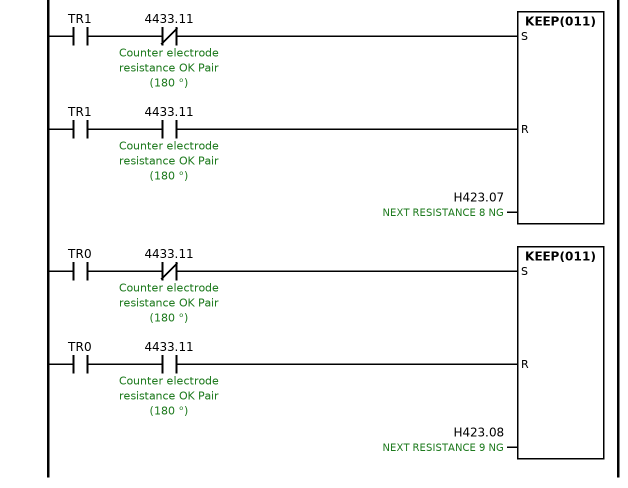
; [picture p408: MainProgram / ST07_RESISTANSE_UNIT, rungs 120-120]
; rung 120
LD 4433.08  ; Counter electrode resistance measurement (180 °)
OUT TR0
AND 4421.01  ; Number of counter electrode resistance 1 *
OUT TR1
ANDNOT 4433.11  ; Counter electrode resistance OK Pair (180 °)
LD TR1
AND 4433.11  ; Counter electrode resistance OK Pair (180 °)
KEEP(011) H423.00  ; NEXT RESISTANCE 1 NG
LD TR0
AND 4421.02  ; Number of adjacent resistances * 2
OUT TR1
ANDNOT 4433.11  ; Counter electrode resistance OK Pair (180 °)
LD TR1
AND 4433.11  ; Counter electrode resistance OK Pair (180 °)
KEEP(011) H423.01  ; NEXT RESISTANCE 2 NG
LD TR0
AND 4421.03  ; Number of adjacent resistances * 3
OUT TR1
ANDNOT 4433.11  ; Counter electrode resistance OK Pair (180 °)
LD TR1
AND 4433.11  ; Counter electrode resistance OK Pair (180 °)
KEEP(011) H423.02  ; NEXT RESISTANCE 3 NG
LD TR0
AND 4421.04  ; Number of adjacent resistances * 4
OUT TR1
ANDNOT 4433.11  ; Counter electrode resistance OK Pair (180 °)
LD TR1
AND 4433.11  ; Counter electrode resistance OK Pair (180 °)
KEEP(011) H423.03  ; NEXT RESISTANCE 4 NG
LD TR0
AND 4421.05  ; Number of adjacent resistances * 5
OUT TR1
ANDNOT 4433.11  ; Counter electrode resistance OK Pair (180 °)
LD TR1
AND 4433.11  ; Counter electrode resistance OK Pair (180 °)
KEEP(011) H423.04  ; NEXT RESISTANCE 5 NG
LD TR0
AND 4421.06  ; Number of adjacent resistances * 6
OUT TR1
ANDNOT 4433.11  ; Counter electrode resistance OK Pair (180 °)
LD TR1
AND 4433.11  ; Counter electrode resistance OK Pair (180 °)
KEEP(011) H423.05  ; NEXT RESISTANCE 6 NG
LD TR0
AND 4421.07  ; Number of adjacent resistances * 7
OUT TR1
ANDNOT 4433.11  ; Counter electrode resistance OK Pair (180 °)
LD TR1
AND 4433.11  ; Counter electrode resistance OK Pair (180 °)
KEEP(011) H423.06  ; NEXT RESISTANCE 7 NG
LD TR0
AND 4421.08  ; Number of adjacent resistances * 8
OUT TR1
ANDNOT 4433.11  ; Counter electrode resistance OK Pair (180 °)
LD TR1
AND 4433.11  ; Counter electrode resistance OK Pair (180 °)
KEEP(011) H423.07  ; NEXT RESISTANCE 8 NG
LD TR0
AND 4421.09  ; Number of adjacent resistances * 9
OUT TR0
ANDNOT 4433.11  ; Counter electrode resistance OK Pair (180 °)
LD TR0
AND 4433.11  ; Counter electrode resistance OK Pair (180 °)
KEEP(011) H423.08  ; NEXT RESISTANCE 9 NG

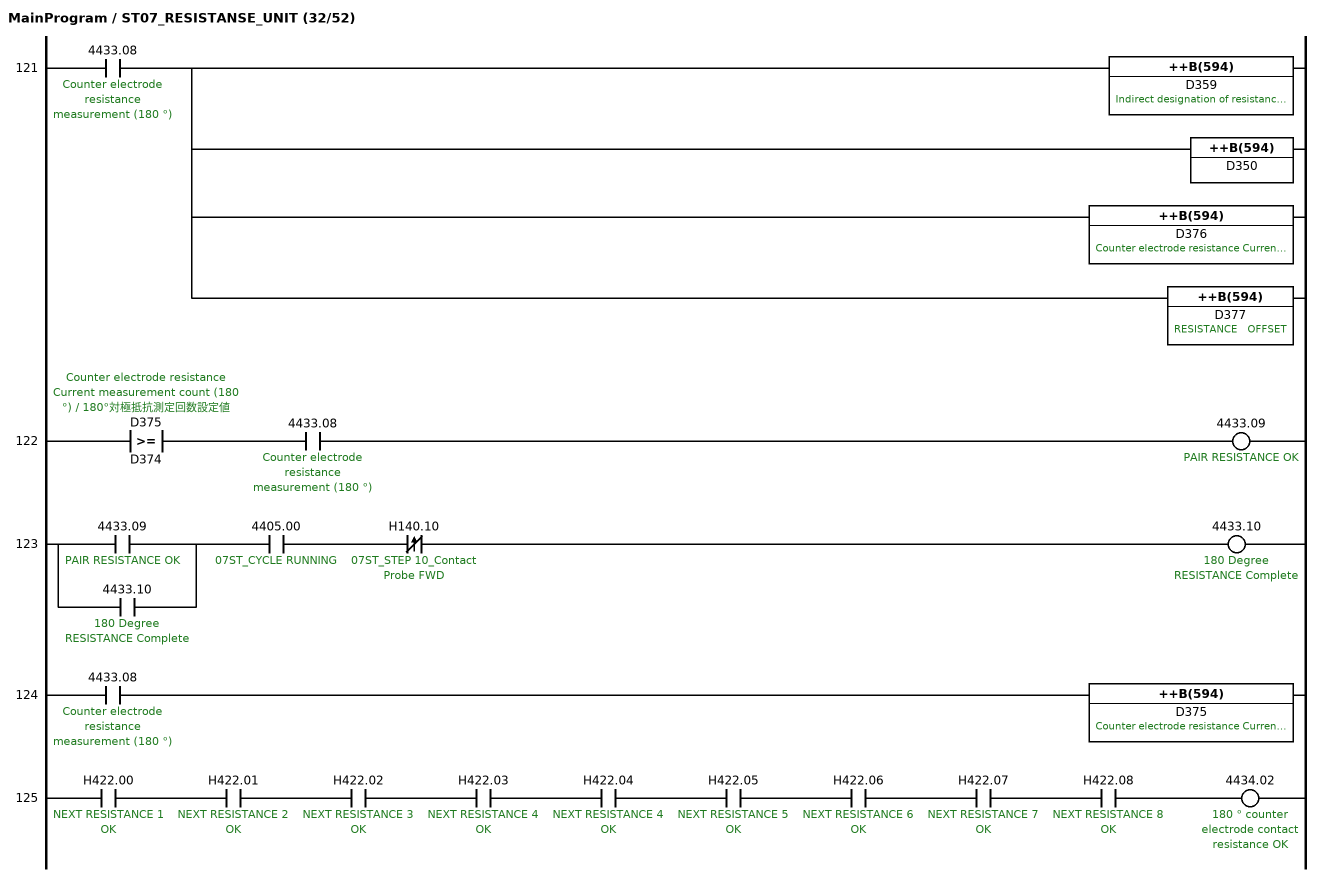
; rung 121
LD 4433.08  ; Counter electrode resistance measurement (180 °)
++B(594) D359  ; Indirect designation of resistance counter electrode data (180 °)  // 
++B(594) D350  // 
++B(594) D376  ; Counter electrode resistance Current measurement count (180 °)  // 
++B(594) D377  ; RESISTANCE　OFFSET  // 
; rung 122
LD>=(325) D375 D374  ; Counter electrode resistance Current measurement count (180 °), 180°対極抵抗測定回数設定値
AND 4433.08  ; Counter electrode resistance measurement (180 °)
OUT 4433.09  ; PAIR RESISTANCE OK
; rung 123
LD 4433.09  ; PAIR RESISTANCE OK
OR 4433.10  ; 180 Degree  RESISTANCE Complete
AND 4405.00  ; 07ST_CYCLE RUNNING
@ANDNOT H140.10  ; 07ST_STEP 10_Contact Probe FWD
OUT 4433.10  ; 180 Degree  RESISTANCE Complete
; rung 124
LD 4433.08  ; Counter electrode resistance measurement (180 °)
++B(594) D375  ; Counter electrode resistance Current measurement count (180 °)  // 
; rung 125
LD H422.00  ; NEXT RESISTANCE 1 OK
AND H422.01  ; NEXT RESISTANCE 2 OK
AND H422.02  ; NEXT RESISTANCE 3 OK
AND H422.03  ; NEXT RESISTANCE 4 OK
AND H422.04  ; NEXT RESISTANCE 4 OK
AND H422.05  ; NEXT RESISTANCE 5 OK
AND H422.06  ; NEXT RESISTANCE 6 OK
AND H422.07  ; NEXT RESISTANCE 7 OK
AND H422.08  ; NEXT RESISTANCE 8 OK
OUT 4434.02  ; 180 ° counter electrode contact resistance OK

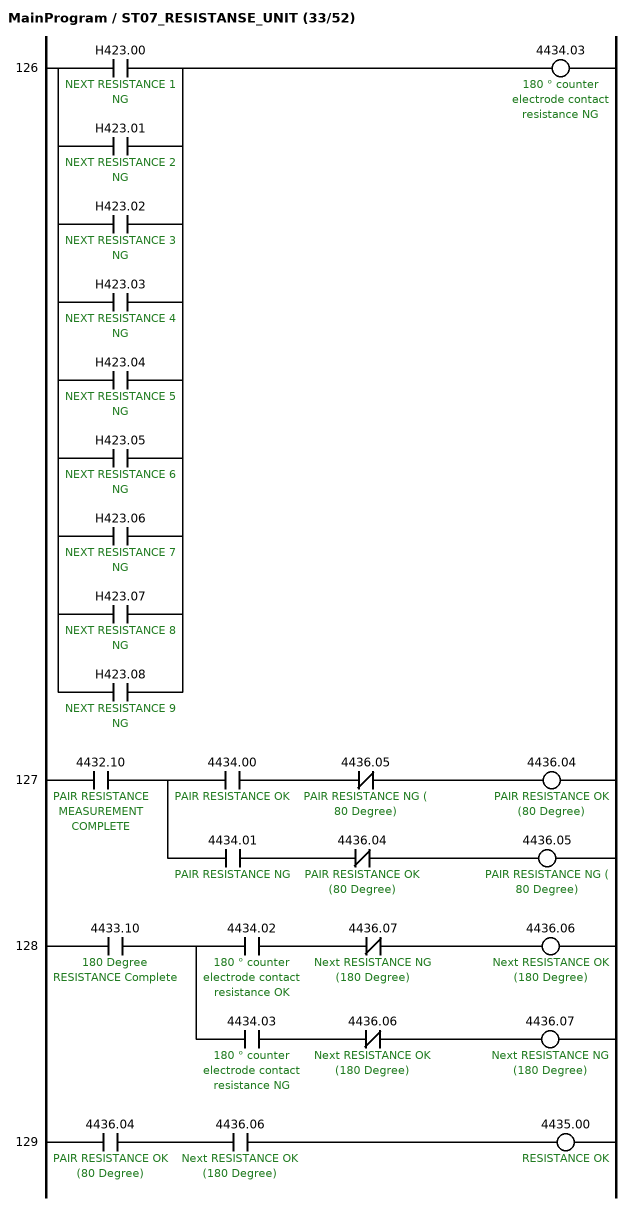
; rung 126
LD H423.00  ; NEXT RESISTANCE 1 NG
OR H423.01  ; NEXT RESISTANCE 2 NG
OR H423.02  ; NEXT RESISTANCE 3 NG
OR H423.03  ; NEXT RESISTANCE 4 NG
OR H423.04  ; NEXT RESISTANCE 5 NG
OR H423.05  ; NEXT RESISTANCE 6 NG
OR H423.06  ; NEXT RESISTANCE 7 NG
OR H423.07  ; NEXT RESISTANCE 8 NG
OR H423.08  ; NEXT RESISTANCE 9 NG
OUT 4434.03  ; 180 ° counter electrode contact resistance NG
; rung 127
LD 4432.10  ; PAIR RESISTANCE MEASUREMENT COMPLETE
OUT TR0
AND 4434.00  ; PAIR RESISTANCE OK
ANDNOT 4436.05  ; PAIR RESISTANCE NG ( 80 Degree)
OUT 4436.04  ; PAIR RESISTANCE OK (80 Degree)
LD TR0
AND 4434.01  ; PAIR RESISTANCE NG
ANDNOT 4436.04  ; PAIR RESISTANCE OK (80 Degree)
OUT 4436.05  ; PAIR RESISTANCE NG ( 80 Degree)
; rung 128
LD 4433.10  ; 180 Degree  RESISTANCE Complete
OUT TR0
AND 4434.02  ; 180 ° counter electrode contact resistance OK
ANDNOT 4436.07  ; Next RESISTANCE NG (180 Degree)
OUT 4436.06  ; Next RESISTANCE OK (180 Degree)
LD TR0
AND 4434.03  ; 180 ° counter electrode contact resistance NG
ANDNOT 4436.06  ; Next RESISTANCE OK (180 Degree)
OUT 4436.07  ; Next RESISTANCE NG (180 Degree)
; rung 129
LD 4436.04  ; PAIR RESISTANCE OK (80 Degree)
AND 4436.06  ; Next RESISTANCE OK (180 Degree)
OUT 4435.00  ; RESISTANCE OK

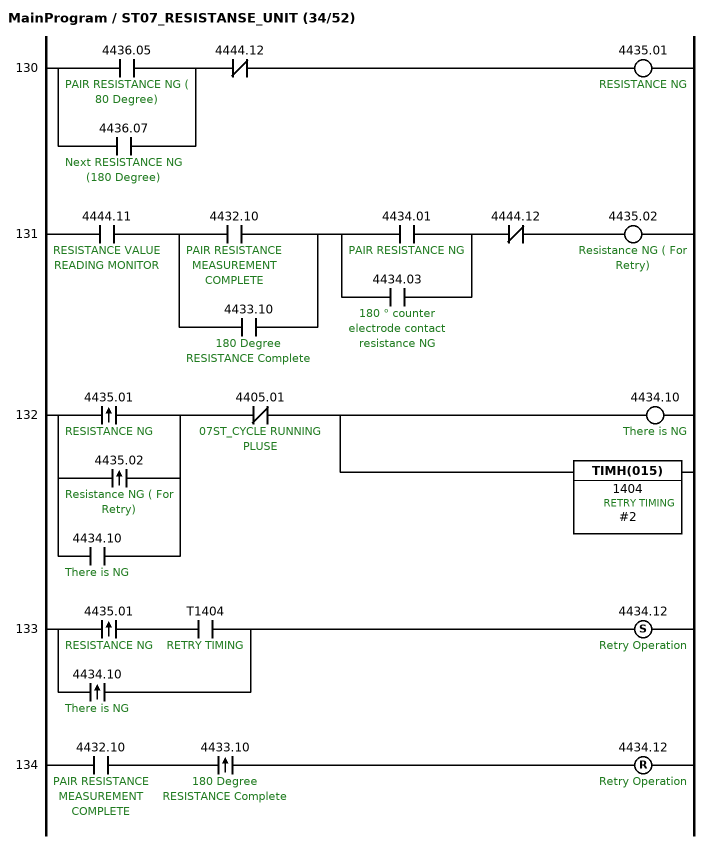
; rung 130
LD 4436.05  ; PAIR RESISTANCE NG ( 80 Degree)
OR 4436.07  ; Next RESISTANCE NG (180 Degree)
ANDNOT 4444.12
OUT 4435.01  ; RESISTANCE NG
; rung 131
LD 4444.11  ; RESISTANCE VALUE READING MONITOR
LD 4432.10  ; PAIR RESISTANCE MEASUREMENT COMPLETE
OR 4433.10  ; 180 Degree  RESISTANCE Complete
ANDLD
LD 4434.01  ; PAIR RESISTANCE NG
OR 4434.03  ; 180 ° counter electrode contact resistance NG
ANDLD
ANDNOT 4444.12
OUT 4435.02  ; Resistance NG ( For Retry)
; rung 132
@LD 4435.01  ; RESISTANCE NG
@OR 4435.02  ; Resistance NG ( For Retry)
OR 4434.10  ; There is NG
ANDNOT 4405.01  ; 07ST_CYCLE RUNNING PLUSE
OUT 4434.10  ; There is NG
TIMH(015) 1404 #2  ; RETRY TIMING
; rung 133
@LD 4435.01  ; RESISTANCE NG
AND T1404  ; RETRY TIMING
@OR 4434.10  ; There is NG
SET 4434.12  ; Retry Operation
; rung 134
LD 4432.10  ; PAIR RESISTANCE MEASUREMENT COMPLETE
@AND 4433.10  ; 180 Degree  RESISTANCE Complete
RSET 4434.12  ; Retry Operation

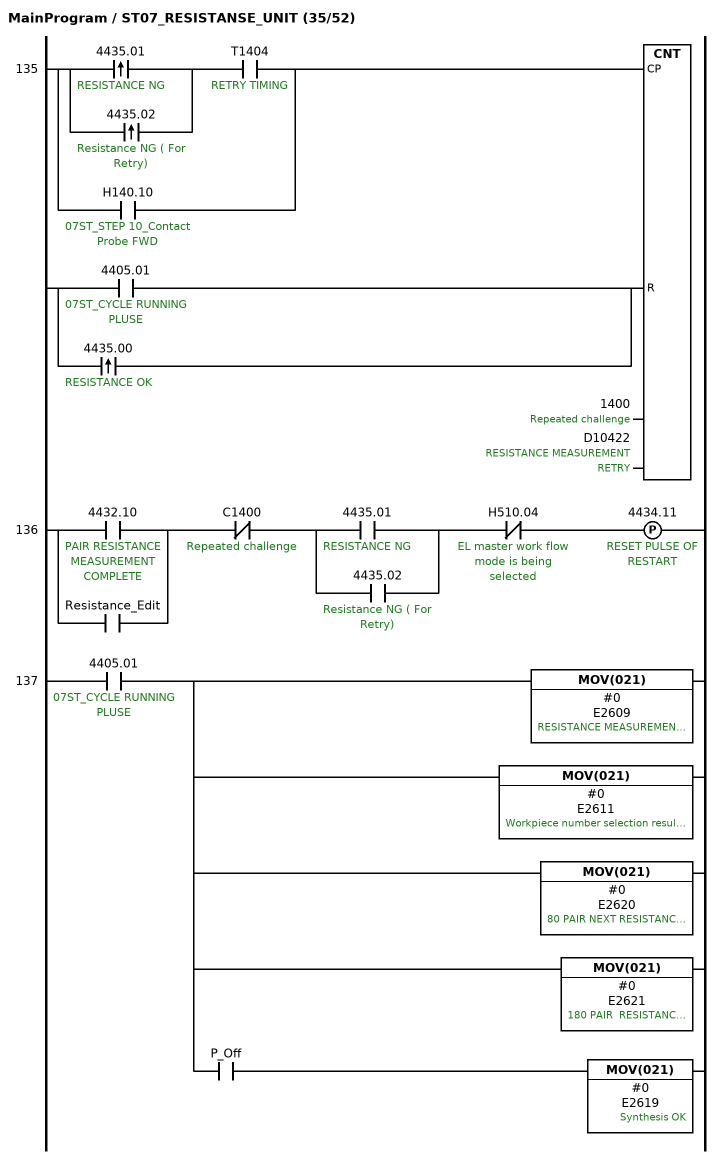
; rung 135
@LD 4435.01  ; RESISTANCE NG
@OR 4435.02  ; Resistance NG ( For Retry)
AND T1404  ; RETRY TIMING
OR H140.10  ; 07ST_STEP 10_Contact Probe FWD
LD 4405.01  ; 07ST_CYCLE RUNNING PLUSE
@OR 4435.00  ; RESISTANCE OK
CNT 1400 D10422  ; RESISTANCE MEASUREMENT RETRY, Repeated challenge
; rung 136
LD 4432.10  ; PAIR RESISTANCE MEASUREMENT COMPLETE
OR Resistance_Edit
ANDNOT C1400  ; Repeated challenge
LD 4435.01  ; RESISTANCE NG
OR 4435.02  ; Resistance NG ( For Retry)
ANDLD
ANDNOT H510.04  ; EL master work flow mode is being selected
DIFU(013) 4434.11  ; RESET PULSE OF RESTART
; rung 137
LD 4405.01  ; 07ST_CYCLE RUNNING PLUSE
MOV(021) #0 E2609  ; RESISTANCE MEASUREMENT JUDGMENT RESULT  (1:OK,2:NG)
MOV(021) #0 E2611  ; Workpiece number selection result (1:OK,2:NG)
MOV(021) #0 E2620  ; 80 PAIR NEXT RESISTANCE MEASUREMENT JUDGMENT RESULT (1:OK,2:NG)
MOV(021) #0 E2621  ; 180 PAIR  RESISTANCE MEASUREMENT JUDGMENT RESULT (1:OK,2:NG)
AND P_Off
MOV(021) #0 E2619  ; Synthesis OK

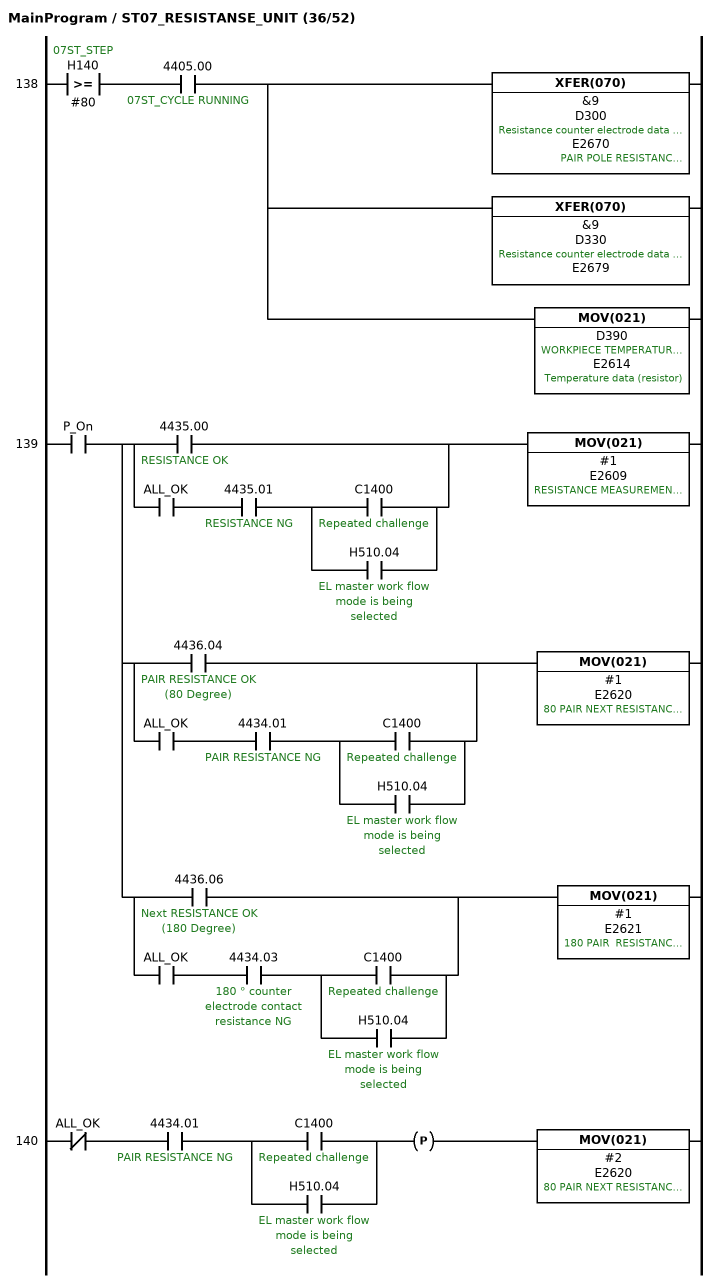
; rung 138
LD>=(325) H140 #80  ; 07ST_STEP
AND 4405.00  ; 07ST_CYCLE RUNNING
XFER(070) &9 D300 E2670  ; Resistance counter electrode data 9 (80 ° counter electrode), PAIR POLE RESISTANCE MEASUREMENT DATA 1
XFER(070) &9 D330 E2679  ; Resistance counter electrode data 1 (180 ° counter electrode)
MOV(021) D390 E2614  ; WORKPIECE TEMPERATURE READING(BCD), Temperature data (resistor)
; rung 139
LD P_On
OUT TR0
LD 4435.00  ; RESISTANCE OK
LD ALL_OK
AND 4435.01  ; RESISTANCE NG
LD C1400  ; Repeated challenge
OR H510.04  ; EL master work flow mode is being selected
ANDLD
ORLD
ANDLD
MOV(021) #1 E2609  ; RESISTANCE MEASUREMENT JUDGMENT RESULT  (1:OK,2:NG)
LD TR0
LD 4436.04  ; PAIR RESISTANCE OK (80 Degree)
LD ALL_OK
AND 4434.01  ; PAIR RESISTANCE NG
LD C1400  ; Repeated challenge
OR H510.04  ; EL master work flow mode is being selected
ANDLD
ORLD
ANDLD
MOV(021) #1 E2620  ; 80 PAIR NEXT RESISTANCE MEASUREMENT JUDGMENT RESULT (1:OK,2:NG)
LD TR0
LD 4436.06  ; Next RESISTANCE OK (180 Degree)
LD ALL_OK
AND 4434.03  ; 180 ° counter electrode contact resistance NG
LD C1400  ; Repeated challenge
OR H510.04  ; EL master work flow mode is being selected
ANDLD
ORLD
ANDLD
MOV(021) #1 E2621  ; 180 PAIR  RESISTANCE MEASUREMENT JUDGMENT RESULT (1:OK,2:NG)
; rung 140
LDNOT ALL_OK
AND 4434.01  ; PAIR RESISTANCE NG
LD C1400  ; Repeated challenge
OR H510.04  ; EL master work flow mode is being selected
ANDLD
UP(521)
MOV(021) #2 E2620  ; 80 PAIR NEXT RESISTANCE MEASUREMENT JUDGMENT RESULT (1:OK,2:NG)

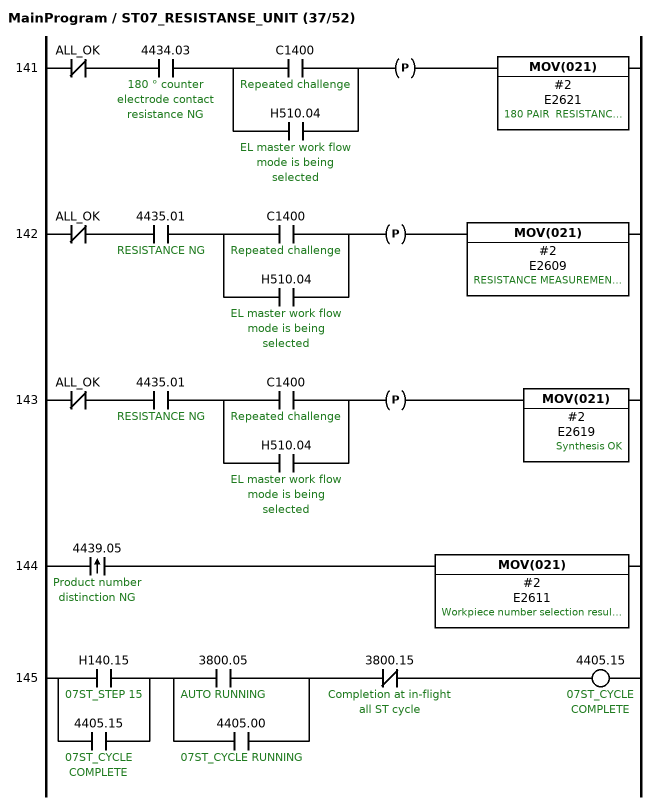
; rung 141
LDNOT ALL_OK
AND 4434.03  ; 180 ° counter electrode contact resistance NG
LD C1400  ; Repeated challenge
OR H510.04  ; EL master work flow mode is being selected
ANDLD
UP(521)
MOV(021) #2 E2621  ; 180 PAIR  RESISTANCE MEASUREMENT JUDGMENT RESULT (1:OK,2:NG)
; rung 142
LDNOT ALL_OK
AND 4435.01  ; RESISTANCE NG
LD C1400  ; Repeated challenge
OR H510.04  ; EL master work flow mode is being selected
ANDLD
UP(521)
MOV(021) #2 E2609  ; RESISTANCE MEASUREMENT JUDGMENT RESULT  (1:OK,2:NG)
; rung 143
LDNOT ALL_OK
AND 4435.01  ; RESISTANCE NG
LD C1400  ; Repeated challenge
OR H510.04  ; EL master work flow mode is being selected
ANDLD
UP(521)
MOV(021) #2 E2619  ; Synthesis OK
; rung 144
@LD 4439.05  ; Product number distinction NG
MOV(021) #2 E2611  ; Workpiece number selection result (1:OK,2:NG)
; rung 145
LD H140.15  ; 07ST_STEP 15
OR 4405.15  ; 07ST_CYCLE COMPLETE
LD 3800.05  ; AUTO RUNNING
OR 4405.00  ; 07ST_CYCLE RUNNING
ANDLD
ANDNOT 3800.15  ; Completion at in-flight all ST cycle
OUT 4405.15  ; 07ST_CYCLE COMPLETE

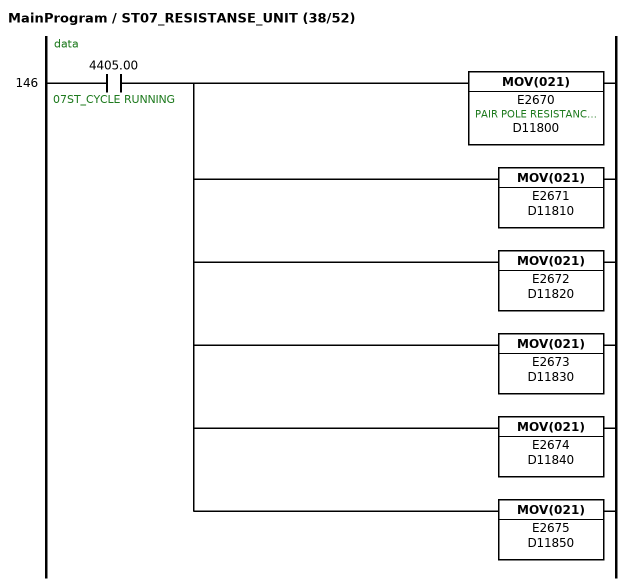
; rung 146: data
LD 4405.00  ; 07ST_CYCLE RUNNING
MOV(021) E2670 D11800  ; PAIR POLE RESISTANCE MEASUREMENT DATA 1
MOV(021) E2671 D11810
MOV(021) E2672 D11820
MOV(021) E2673 D11830
MOV(021) E2674 D11840
MOV(021) E2675 D11850

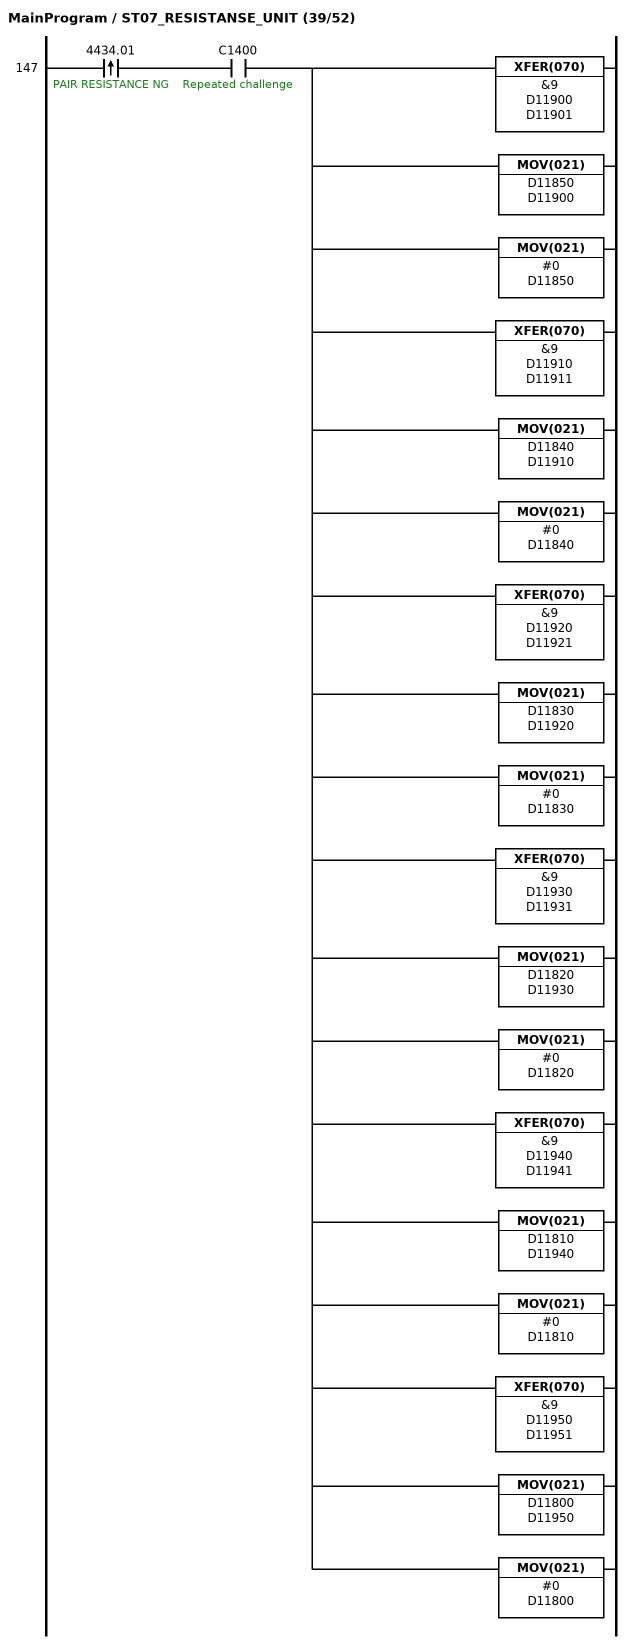
; rung 147
@LD 4434.01  ; PAIR RESISTANCE NG
AND C1400  ; Repeated challenge
XFER(070) &9 D11900 D11901
MOV(021) D11850 D11900
MOV(021) #0 D11850
XFER(070) &9 D11910 D11911
MOV(021) D11840 D11910
MOV(021) #0 D11840
XFER(070) &9 D11920 D11921
MOV(021) D11830 D11920
MOV(021) #0 D11830
XFER(070) &9 D11930 D11931
MOV(021) D11820 D11930
MOV(021) #0 D11820
XFER(070) &9 D11940 D11941
MOV(021) D11810 D11940
MOV(021) #0 D11810
XFER(070) &9 D11950 D11951
MOV(021) D11800 D11950
MOV(021) #0 D11800

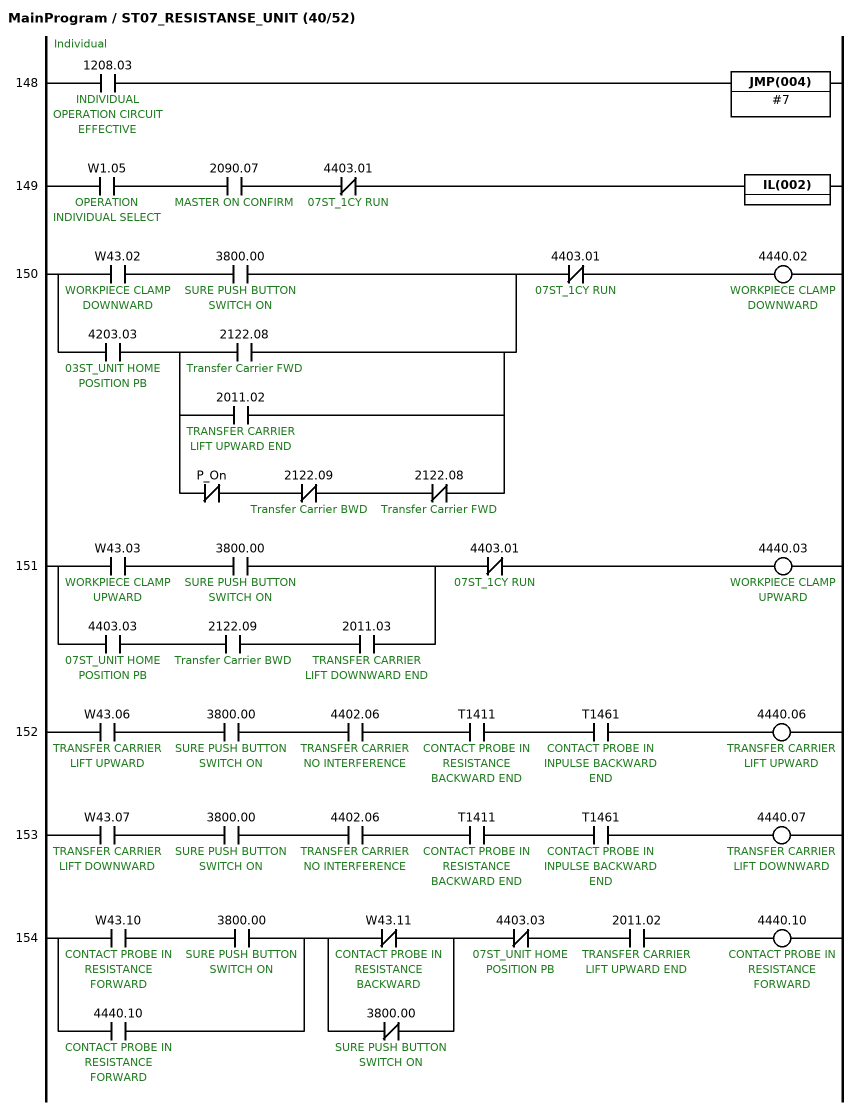
; rung 148: Individual
LD 1208.03  ; INDIVIDUAL OPERATION CIRCUIT EFFECTIVE
JMP(004) #7
; rung 149
LD W1.05  ; OPERATION INDIVIDUAL SELECT
AND 2090.07  ; MASTER ON CONFIRM
ANDNOT 4403.01  ; 07ST_1CY RUN
IL(002)
; rung 150
LD W43.02  ; WORKPIECE CLAMP DOWNWARD
AND 3800.00  ; SURE PUSH BUTTON SWITCH ON
LD 4203.03  ; 03ST_UNIT HOME POSITION PB
LD 2122.08  ; Transfer Carrier FWD
OR 2011.02  ; TRANSFER CARRIER LIFT UPWARD END
LDNOT P_On
ANDNOT 2122.09  ; Transfer Carrier BWD
ANDNOT 2122.08  ; Transfer Carrier FWD
ORLD
ANDLD
ORLD
ANDNOT 4403.01  ; 07ST_1CY RUN
OUT 4440.02  ; WORKPIECE CLAMP DOWNWARD
; rung 151
LD W43.03  ; WORKPIECE CLAMP UPWARD
AND 3800.00  ; SURE PUSH BUTTON SWITCH ON
LD 4403.03  ; 07ST_UNIT HOME POSITION PB
AND 2122.09  ; Transfer Carrier BWD
AND 2011.03  ; TRANSFER CARRIER LIFT DOWNWARD END
ORLD
ANDNOT 4403.01  ; 07ST_1CY RUN
OUT 4440.03  ; WORKPIECE CLAMP UPWARD
; rung 152
LD W43.06  ; TRANSFER CARRIER LIFT UPWARD
AND 3800.00  ; SURE PUSH BUTTON SWITCH ON
AND 4402.06  ; TRANSFER CARRIER NO INTERFERENCE
AND T1411  ; CONTACT PROBE IN RESISTANCE BACKWARD END
AND T1461  ; CONTACT PROBE IN INPULSE BACKWARD END
OUT 4440.06  ; TRANSFER CARRIER LIFT UPWARD
; rung 153
LD W43.07  ; TRANSFER CARRIER LIFT DOWNWARD
AND 3800.00  ; SURE PUSH BUTTON SWITCH ON
AND 4402.06  ; TRANSFER CARRIER NO INTERFERENCE
AND T1411  ; CONTACT PROBE IN RESISTANCE BACKWARD END
AND T1461  ; CONTACT PROBE IN INPULSE BACKWARD END
OUT 4440.07  ; TRANSFER CARRIER LIFT DOWNWARD
; rung 154
LD W43.10  ; CONTACT PROBE IN RESISTANCE FORWARD
AND 3800.00  ; SURE PUSH BUTTON SWITCH ON
OR 4440.10  ; CONTACT PROBE IN RESISTANCE FORWARD
LDNOT W43.11  ; CONTACT PROBE IN RESISTANCE BACKWARD
ORNOT 3800.00  ; SURE PUSH BUTTON SWITCH ON
ANDLD
ANDNOT 4403.03  ; 07ST_UNIT HOME POSITION PB
AND 2011.02  ; TRANSFER CARRIER LIFT UPWARD END
OUT 4440.10  ; CONTACT PROBE IN RESISTANCE FORWARD

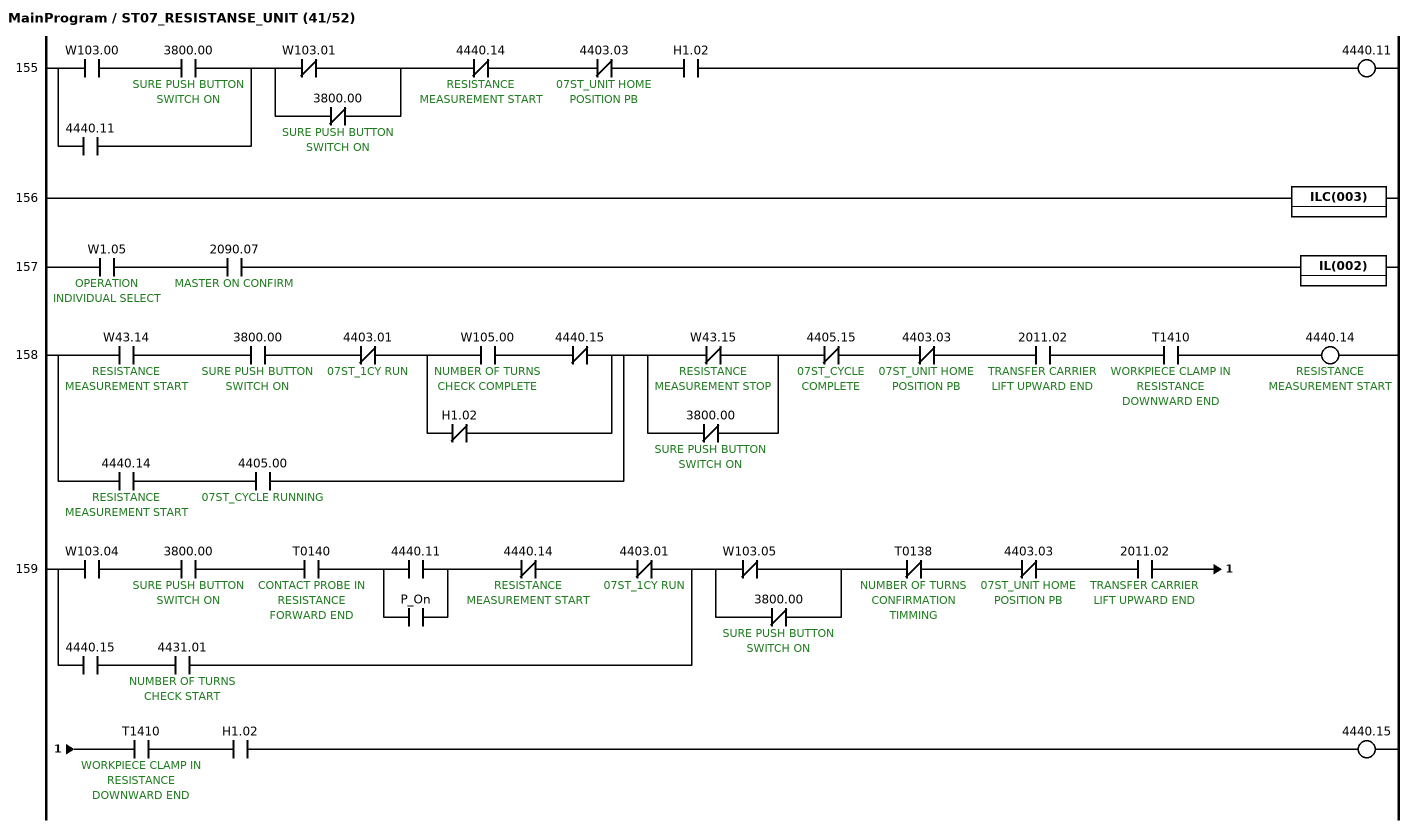
; rung 155
LD W103.00
AND 3800.00  ; SURE PUSH BUTTON SWITCH ON
OR 4440.11
LDNOT W103.01
ORNOT 3800.00  ; SURE PUSH BUTTON SWITCH ON
ANDLD
ANDNOT 4440.14  ; RESISTANCE MEASUREMENT START
ANDNOT 4403.03  ; 07ST_UNIT HOME POSITION PB
AND H1.02
OUT 4440.11
; rung 156
ILC(003)
; rung 157
LD W1.05  ; OPERATION INDIVIDUAL SELECT
AND 2090.07  ; MASTER ON CONFIRM
IL(002)
; rung 158
LD W43.14  ; RESISTANCE MEASUREMENT START
AND 3800.00  ; SURE PUSH BUTTON SWITCH ON
ANDNOT 4403.01  ; 07ST_1CY RUN
LD W105.00  ; NUMBER OF TURNS CHECK COMPLETE
ANDNOT 4440.15
ORNOT H1.02
ANDLD
LD 4440.14  ; RESISTANCE MEASUREMENT START
AND 4405.00  ; 07ST_CYCLE RUNNING
ORLD
LDNOT W43.15  ; RESISTANCE MEASUREMENT STOP
ORNOT 3800.00  ; SURE PUSH BUTTON SWITCH ON
ANDLD
ANDNOT 4405.15  ; 07ST_CYCLE COMPLETE
ANDNOT 4403.03  ; 07ST_UNIT HOME POSITION PB
AND 2011.02  ; TRANSFER CARRIER LIFT UPWARD END
AND T1410  ; WORKPIECE CLAMP IN RESISTANCE DOWNWARD END
OUT 4440.14  ; RESISTANCE MEASUREMENT START
; rung 159
LD W103.04
AND 3800.00  ; SURE PUSH BUTTON SWITCH ON
AND T0140  ; CONTACT PROBE IN RESISTANCE FORWARD END
LD 4440.11
OR P_On
ANDLD
ANDNOT 4440.14  ; RESISTANCE MEASUREMENT START
ANDNOT 4403.01  ; 07ST_1CY RUN
LD 4440.15
AND 4431.01  ; NUMBER OF TURNS CHECK START
ORLD
LDNOT W103.05
ORNOT 3800.00  ; SURE PUSH BUTTON SWITCH ON
ANDLD
ANDNOT T0138  ; NUMBER OF TURNS CONFIRMATION TIMMING
ANDNOT 4403.03  ; 07ST_UNIT HOME POSITION PB
AND 2011.02  ; TRANSFER CARRIER LIFT UPWARD END
AND T1410  ; WORKPIECE CLAMP IN RESISTANCE DOWNWARD END
AND H1.02
OUT 4440.15

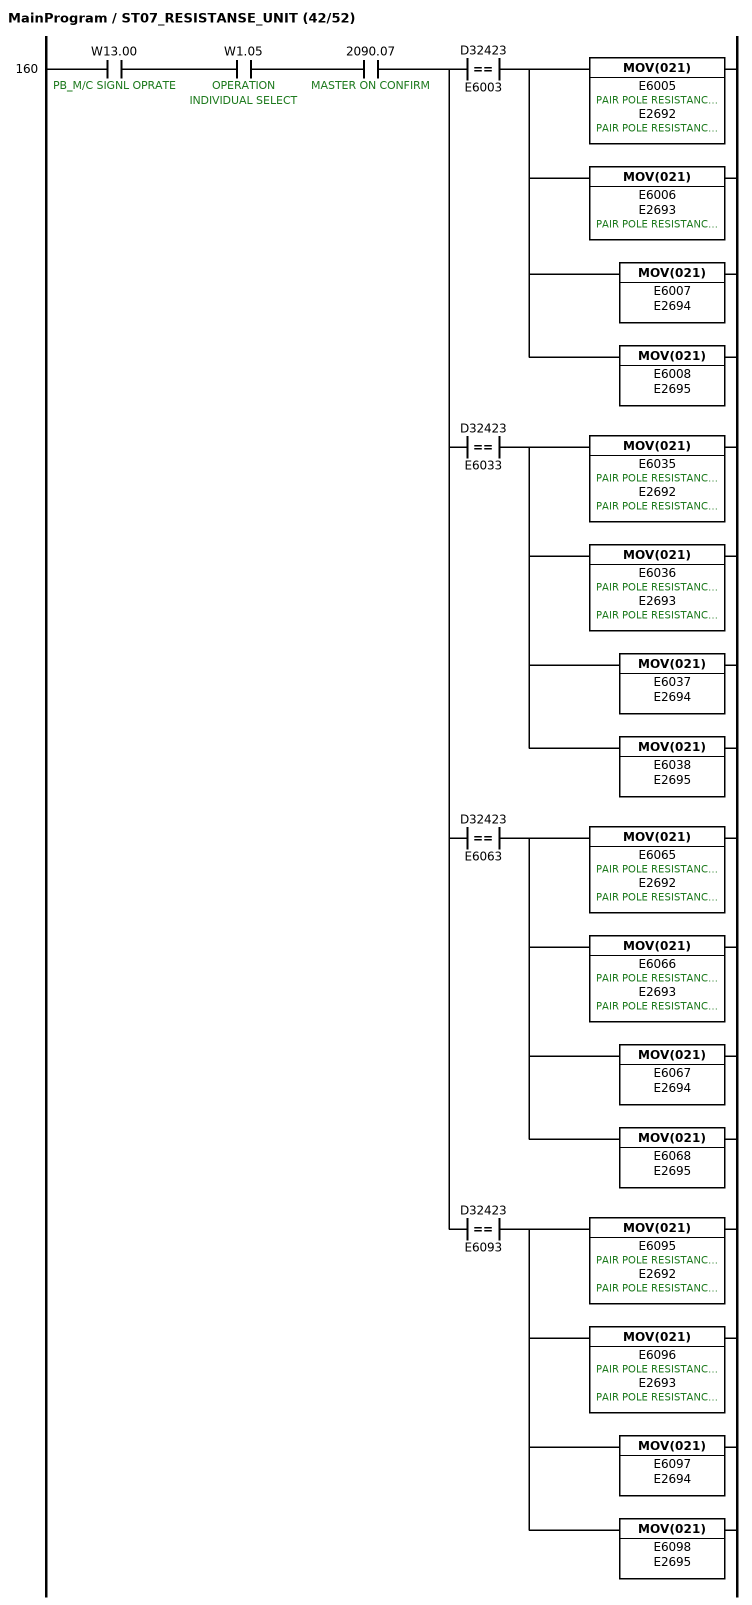
; rung 160
LD W13.00  ; PB_M/C SIGNL OPRATE
AND W1.05  ; OPERATION INDIVIDUAL SELECT
AND 2090.07  ; MASTER ON CONFIRM
OUT TR0
AND=(300) D32423 E6003
MOV(021) E6005 E2692  ; PAIR POLE RESISTANCE MEASUREMENT DATA 1, PAIR POLE RESISTANCE SPECIFICATION MINIMUM VALUE
MOV(021) E6006 E2693  ; PAIR POLE RESISTANCE SPECIFICATION MAXIMUM VALUE
MOV(021) E6007 E2694
MOV(021) E6008 E2695
LD TR0
AND=(300) D32423 E6033
MOV(021) E6035 E2692  ; PAIR POLE RESISTANCE MEASUREMENT DATA 1, PAIR POLE RESISTANCE SPECIFICATION MINIMUM VALUE
MOV(021) E6036 E2693  ; PAIR POLE RESISTANCE MEASUREMENT DATA 1, PAIR POLE RESISTANCE SPECIFICATION MAXIMUM VALUE
MOV(021) E6037 E2694
MOV(021) E6038 E2695
LD TR0
AND=(300) D32423 E6063
MOV(021) E6065 E2692  ; PAIR POLE RESISTANCE SPECIFICATION MINIMUM VALUE
MOV(021) E6066 E2693  ; PAIR POLE RESISTANCE SPECIFICATION MAXIMUM VALUE
MOV(021) E6067 E2694
MOV(021) E6068 E2695
LD TR0
AND=(300) D32423 E6093
MOV(021) E6095 E2692  ; PAIR POLE RESISTANCE SPECIFICATION MINIMUM VALUE
MOV(021) E6096 E2693  ; PAIR POLE RESISTANCE SPECIFICATION MAXIMUM VALUE
MOV(021) E6097 E2694
MOV(021) E6098 E2695

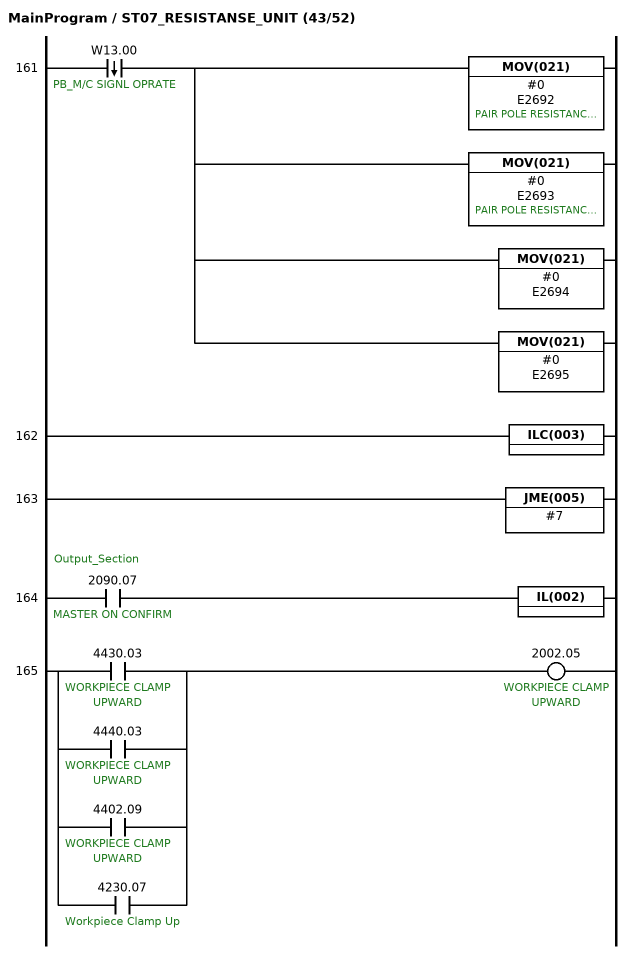
; rung 161
%LD W13.00  ; PB_M/C SIGNL OPRATE
MOV(021) #0 E2692  ; PAIR POLE RESISTANCE SPECIFICATION MINIMUM VALUE
MOV(021) #0 E2693  ; PAIR POLE RESISTANCE SPECIFICATION MAXIMUM VALUE
MOV(021) #0 E2694
MOV(021) #0 E2695
; rung 162
ILC(003)
; rung 163
JME(005) #7
; rung 164: Output_Section
LD 2090.07  ; MASTER ON CONFIRM
IL(002)
; rung 165
LD 4430.03  ; WORKPIECE CLAMP UPWARD
OR 4440.03  ; WORKPIECE CLAMP UPWARD
OR 4402.09  ; WORKPIECE CLAMP UPWARD
OR 4230.07  ; Workpiece Clamp Up
OUT 2002.05  ; WORKPIECE CLAMP UPWARD

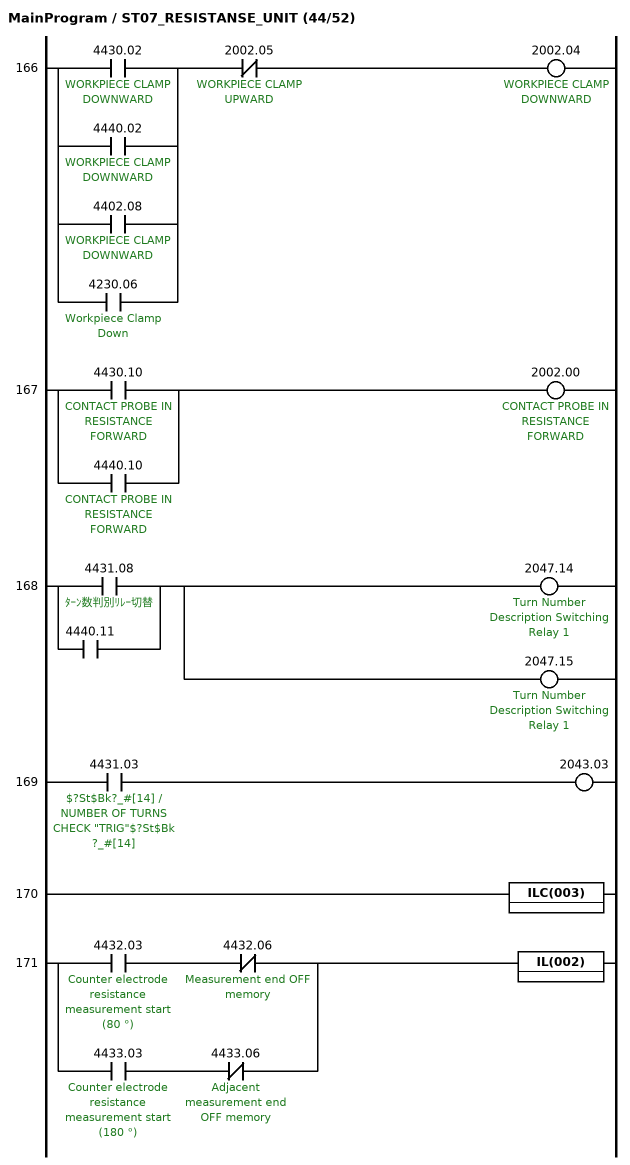
; rung 166
LD 4430.02  ; WORKPIECE CLAMP DOWNWARD
OR 4440.02  ; WORKPIECE CLAMP DOWNWARD
OR 4402.08  ; WORKPIECE CLAMP DOWNWARD
OR 4230.06  ; Workpiece Clamp Down
ANDNOT 2002.05  ; WORKPIECE CLAMP UPWARD
OUT 2002.04  ; WORKPIECE CLAMP DOWNWARD
; rung 167
LD 4430.10  ; CONTACT PROBE IN RESISTANCE FORWARD
OR 4440.10  ; CONTACT PROBE IN RESISTANCE FORWARD
OUT 2002.00  ; CONTACT PROBE IN RESISTANCE FORWARD
; rung 168
LD 4431.08  ; ﾀｰﾝ数判別ﾘﾚｰ切替
OR 4440.11
OUT 2047.14  ; Turn Number Description Switching Relay 1
OUT 2047.15  ; Turn Number Description Switching Relay 1
; rung 169
LD 4431.03  ; $?St$Bk?_#[14] / NUMBER OF TURNS CHECK "TRIG"$?St$Bk?_#[14]
OUT 2043.03
; rung 170
ILC(003)
; rung 171
LD 4432.03  ; Counter electrode resistance measurement start (80 °)
ANDNOT 4432.06  ; Measurement end OFF memory
LD 4433.03  ; Counter electrode resistance measurement start (180 °)
ANDNOT 4433.06  ; Adjacent measurement end OFF memory
ORLD
IL(002)

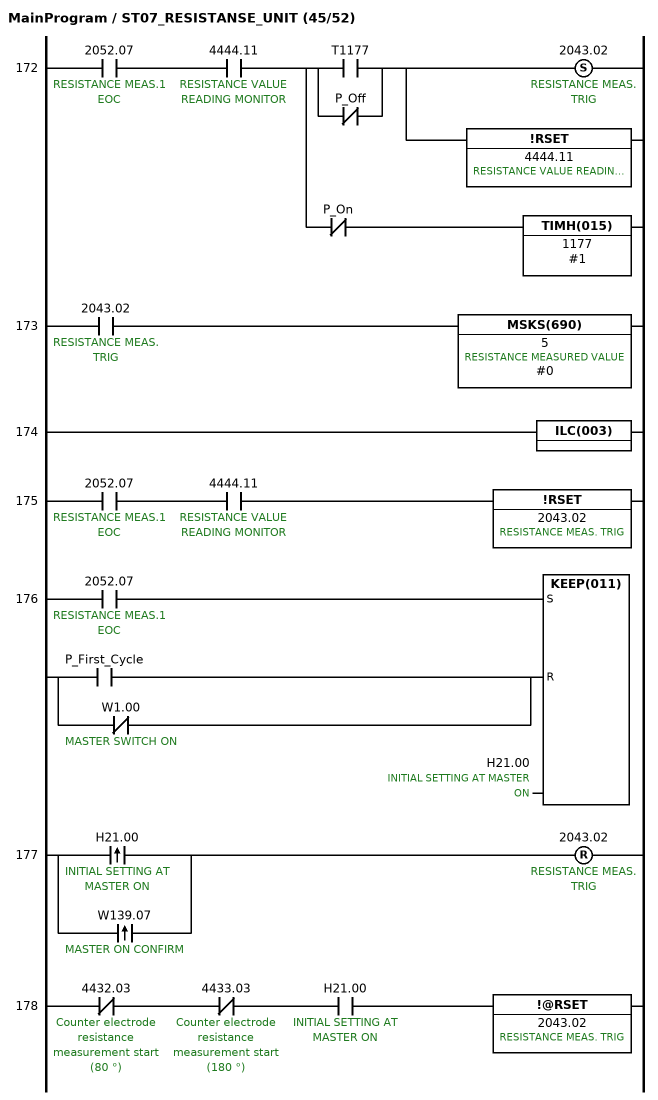
; rung 172
LD 2052.07  ; RESISTANCE MEAS.1 EOC
AND 4444.11  ; RESISTANCE VALUE READING MONITOR
OUT TR0
LD T1177
ORNOT P_Off
ANDLD
SET 2043.02  ; RESISTANCE MEAS. TRIG
!RSET 4444.11  ; RESISTANCE VALUE READING MONITOR
LD TR0
ANDNOT P_On
TIMH(015) 1177 #1
; rung 173
LD 2043.02  ; RESISTANCE MEAS. TRIG
MSKS(690) 5 #0  ; RESISTANCE MEASURED VALUE  // 
; rung 174
ILC(003)
; rung 175
LD 2052.07  ; RESISTANCE MEAS.1 EOC
AND 4444.11  ; RESISTANCE VALUE READING MONITOR
!RSET 2043.02  ; RESISTANCE MEAS. TRIG
; rung 176
LD 2052.07  ; RESISTANCE MEAS.1 EOC
LD P_First_Cycle
ORNOT W1.00  ; MASTER SWITCH ON
KEEP(011) H21.00  ; INITIAL SETTING AT MASTER ON
; rung 177
@LD H21.00  ; INITIAL SETTING AT MASTER ON
@OR W139.07  ; MASTER ON CONFIRM
RSET 2043.02  ; RESISTANCE MEAS. TRIG
; rung 178
LDNOT 4432.03  ; Counter electrode resistance measurement start (80 °)
ANDNOT 4433.03  ; Counter electrode resistance measurement start (180 °)
AND H21.00  ; INITIAL SETTING AT MASTER ON
!@RSET 2043.02  ; RESISTANCE MEAS. TRIG

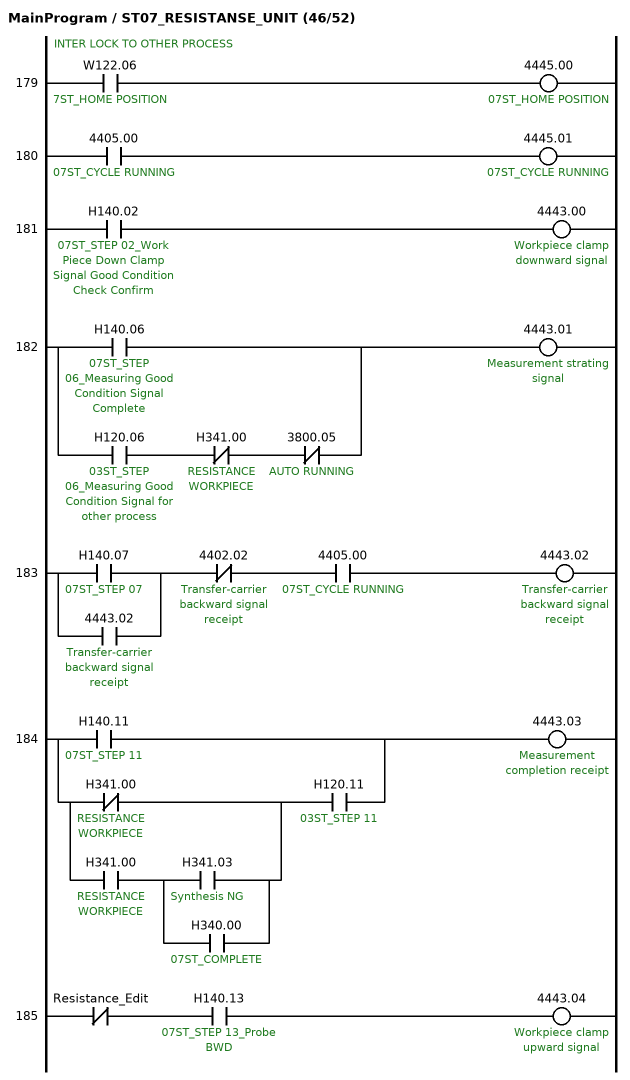
; rung 179: INTER LOCK TO OTHER PROCESS
LD W122.06  ; 7ST_HOME POSITION
OUT 4445.00  ; 07ST_HOME POSITION
; rung 180
LD 4405.00  ; 07ST_CYCLE RUNNING
OUT 4445.01  ; 07ST_CYCLE RUNNING
; rung 181
LD H140.02  ; 07ST_STEP 02_Work Piece Down Clamp Signal Good Condition Check Confirm
OUT 4443.00  ; Workpiece clamp downward signal
; rung 182
LD H140.06  ; 07ST_STEP 06_Measuring Good Condition Signal Complete
LD H120.06  ; 03ST_STEP 06_Measuring Good Condition Signal for other process
ANDNOT H341.00  ; RESISTANCE WORKPIECE
ANDNOT 3800.05  ; AUTO RUNNING
ORLD
OUT 4443.01  ; Measurement strating signal
; rung 183
LD H140.07  ; 07ST_STEP 07
OR 4443.02  ; Transfer-carrier backward signal receipt
ANDNOT 4402.02  ; Transfer-carrier backward signal receipt
AND 4405.00  ; 07ST_CYCLE RUNNING
OUT 4443.02  ; Transfer-carrier backward signal receipt
; rung 184
LD H140.11  ; 07ST_STEP 11
LDNOT H341.00  ; RESISTANCE WORKPIECE
LD H341.00  ; RESISTANCE WORKPIECE
LD H341.03  ; Synthesis NG
OR H340.00  ; 07ST_COMPLETE
ANDLD
ORLD
AND H120.11  ; 03ST_STEP 11
ORLD
OUT 4443.03  ; Measurement completion receipt
; rung 185
LDNOT Resistance_Edit
AND H140.13  ; 07ST_STEP 13_Probe BWD
OUT 4443.04  ; Workpiece clamp upward signal

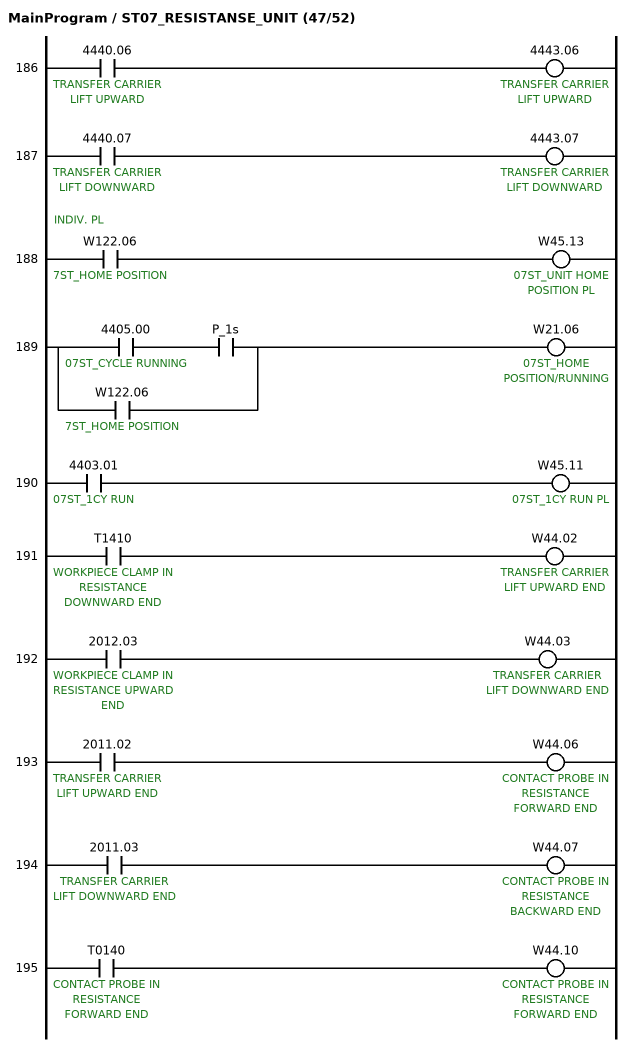
; rung 186
LD 4440.06  ; TRANSFER CARRIER LIFT UPWARD
OUT 4443.06  ; TRANSFER CARRIER LIFT UPWARD
; rung 187
LD 4440.07  ; TRANSFER CARRIER LIFT DOWNWARD
OUT 4443.07  ; TRANSFER CARRIER LIFT DOWNWARD
; rung 188: INDIV. PL
LD W122.06  ; 7ST_HOME POSITION
OUT W45.13  ; 07ST_UNIT HOME POSITION PL
; rung 189
LD 4405.00  ; 07ST_CYCLE RUNNING
AND P_1s
OR W122.06  ; 7ST_HOME POSITION
OUT W21.06  ; 07ST_HOME POSITION/RUNNING
; rung 190
LD 4403.01  ; 07ST_1CY RUN
OUT W45.11  ; 07ST_1CY RUN PL
; rung 191
LD T1410  ; WORKPIECE CLAMP IN RESISTANCE DOWNWARD END
OUT W44.02  ; TRANSFER CARRIER LIFT UPWARD END
; rung 192
LD 2012.03  ; WORKPIECE CLAMP IN RESISTANCE UPWARD END
OUT W44.03  ; TRANSFER CARRIER LIFT DOWNWARD END
; rung 193
LD 2011.02  ; TRANSFER CARRIER LIFT UPWARD END
OUT W44.06  ; CONTACT PROBE IN RESISTANCE FORWARD END
; rung 194
LD 2011.03  ; TRANSFER CARRIER LIFT DOWNWARD END
OUT W44.07  ; CONTACT PROBE IN RESISTANCE BACKWARD END
; rung 195
LD T0140  ; CONTACT PROBE IN RESISTANCE FORWARD END
OUT W44.10  ; CONTACT PROBE IN RESISTANCE FORWARD END

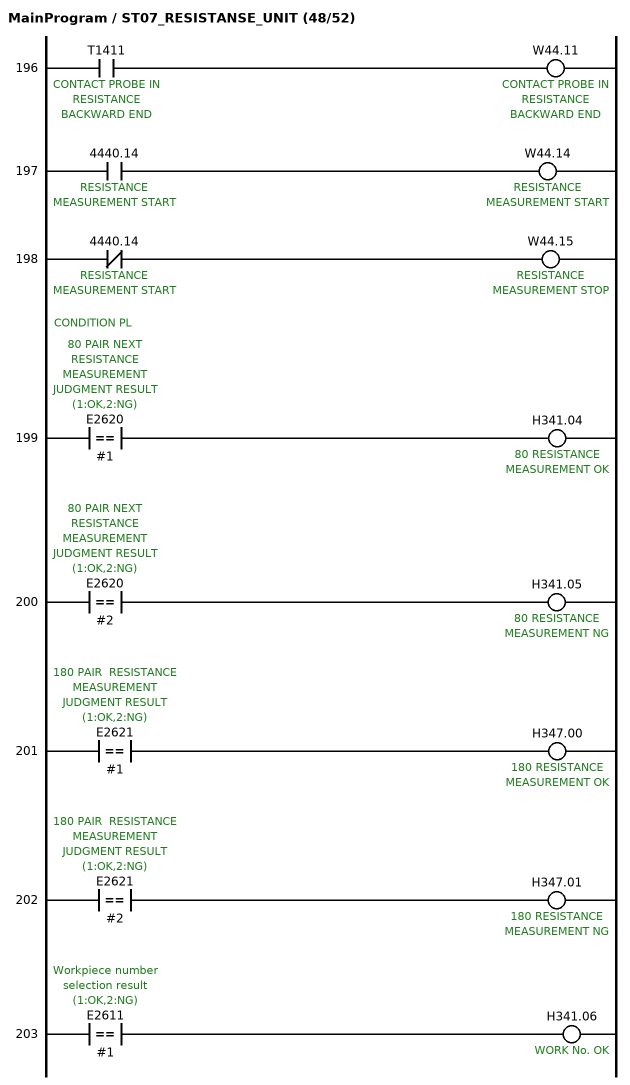
; rung 196
LD T1411  ; CONTACT PROBE IN RESISTANCE BACKWARD END
OUT W44.11  ; CONTACT PROBE IN RESISTANCE BACKWARD END
; rung 197
LD 4440.14  ; RESISTANCE MEASUREMENT START
OUT W44.14  ; RESISTANCE MEASUREMENT START
; rung 198
LDNOT 4440.14  ; RESISTANCE MEASUREMENT START
OUT W44.15  ; RESISTANCE MEASUREMENT STOP
; rung 199: CONDITION PL
LD=(300) E2620 #1  ; 80 PAIR NEXT RESISTANCE MEASUREMENT JUDGMENT RESULT (1:OK,2:NG)
OUT H341.04  ; 80 RESISTANCE MEASUREMENT OK
; rung 200
LD=(300) E2620 #2  ; 80 PAIR NEXT RESISTANCE MEASUREMENT JUDGMENT RESULT (1:OK,2:NG)
OUT H341.05  ; 80 RESISTANCE MEASUREMENT NG
; rung 201
LD=(300) E2621 #1  ; 180 PAIR  RESISTANCE MEASUREMENT JUDGMENT RESULT (1:OK,2:NG)
OUT H347.00  ; 180 RESISTANCE MEASUREMENT OK
; rung 202
LD=(300) E2621 #2  ; 180 PAIR  RESISTANCE MEASUREMENT JUDGMENT RESULT (1:OK,2:NG)
OUT H347.01  ; 180 RESISTANCE MEASUREMENT NG
; rung 203
LD=(300) E2611 #1  ; Workpiece number selection result (1:OK,2:NG)
OUT H341.06  ; WORK No. OK

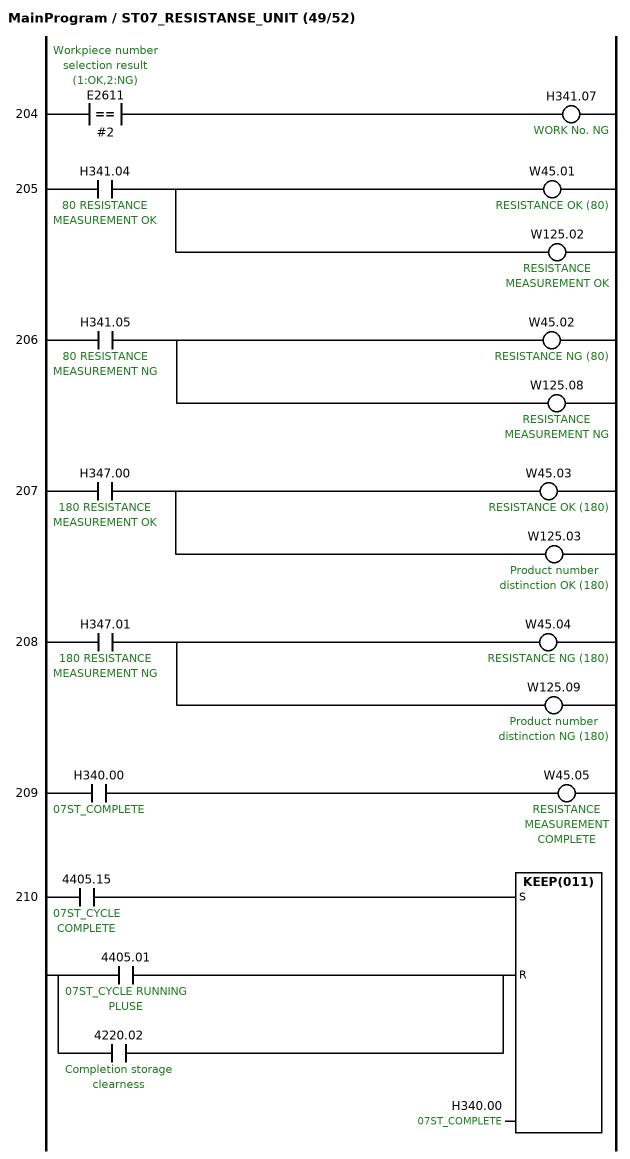
; rung 204
LD=(300) E2611 #2  ; Workpiece number selection result (1:OK,2:NG)
OUT H341.07  ; WORK No. NG
; rung 205
LD H341.04  ; 80 RESISTANCE MEASUREMENT OK
OUT W45.01  ; RESISTANCE OK (80)
OUT W125.02  ; RESISTANCE MEASUREMENT OK
; rung 206
LD H341.05  ; 80 RESISTANCE MEASUREMENT NG
OUT W45.02  ; RESISTANCE NG (80)
OUT W125.08  ; RESISTANCE MEASUREMENT NG
; rung 207
LD H347.00  ; 180 RESISTANCE MEASUREMENT OK
OUT W45.03  ; RESISTANCE OK (180)
OUT W125.03  ; Product number distinction OK (180)
; rung 208
LD H347.01  ; 180 RESISTANCE MEASUREMENT NG
OUT W45.04  ; RESISTANCE NG (180)
OUT W125.09  ; Product number distinction NG (180)
; rung 209
LD H340.00  ; 07ST_COMPLETE
OUT W45.05  ; RESISTANCE MEASUREMENT COMPLETE
; rung 210
LD 4405.15  ; 07ST_CYCLE COMPLETE
LD 4405.01  ; 07ST_CYCLE RUNNING PLUSE
OR 4220.02  ; Completion storage clearness
KEEP(011) H340.00  ; 07ST_COMPLETE

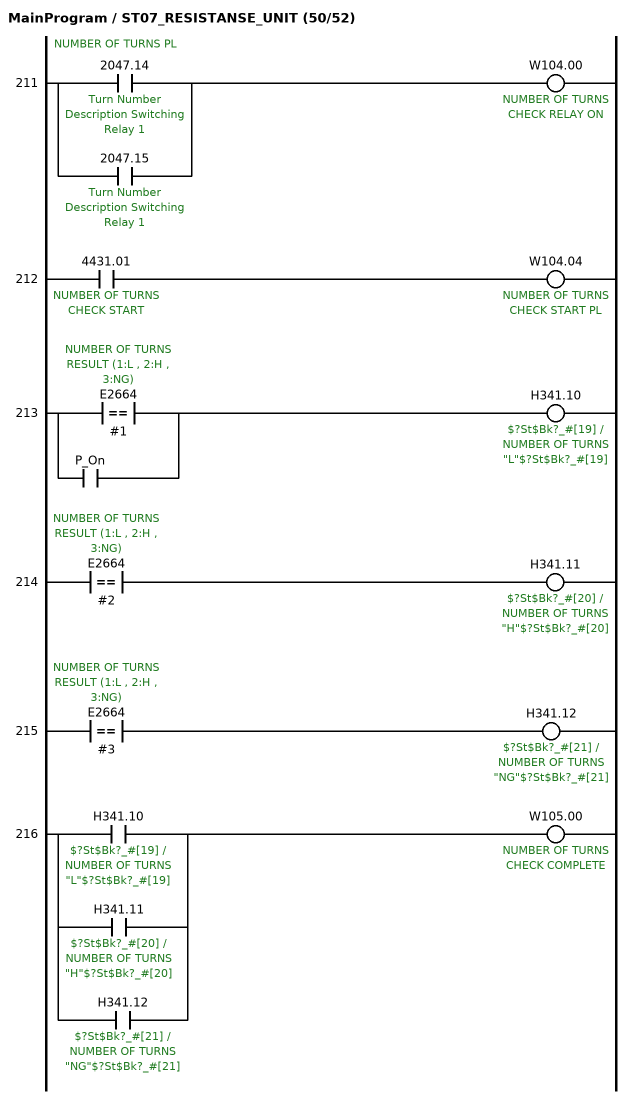
; rung 211: NUMBER OF TURNS PL
LD 2047.14  ; Turn Number Description Switching Relay 1
OR 2047.15  ; Turn Number Description Switching Relay 1
OUT W104.00  ; NUMBER OF TURNS CHECK RELAY ON
; rung 212
LD 4431.01  ; NUMBER OF TURNS CHECK START
OUT W104.04  ; NUMBER OF TURNS CHECK START PL
; rung 213
LD=(300) E2664 #1  ; NUMBER OF TURNS RESULT (1:L , 2:H , 3:NG)
OR P_On
OUT H341.10  ; $?St$Bk?_#[19] / NUMBER OF TURNS "L"$?St$Bk?_#[19]
; rung 214
LD=(300) E2664 #2  ; NUMBER OF TURNS RESULT (1:L , 2:H , 3:NG)
OUT H341.11  ; $?St$Bk?_#[20] / NUMBER OF TURNS "H"$?St$Bk?_#[20]
; rung 215
LD=(300) E2664 #3  ; NUMBER OF TURNS RESULT (1:L , 2:H , 3:NG)
OUT H341.12  ; $?St$Bk?_#[21] / NUMBER OF TURNS "NG"$?St$Bk?_#[21]
; rung 216
LD H341.10  ; $?St$Bk?_#[19] / NUMBER OF TURNS "L"$?St$Bk?_#[19]
OR H341.11  ; $?St$Bk?_#[20] / NUMBER OF TURNS "H"$?St$Bk?_#[20]
OR H341.12  ; $?St$Bk?_#[21] / NUMBER OF TURNS "NG"$?St$Bk?_#[21]
OUT W105.00  ; NUMBER OF TURNS CHECK COMPLETE

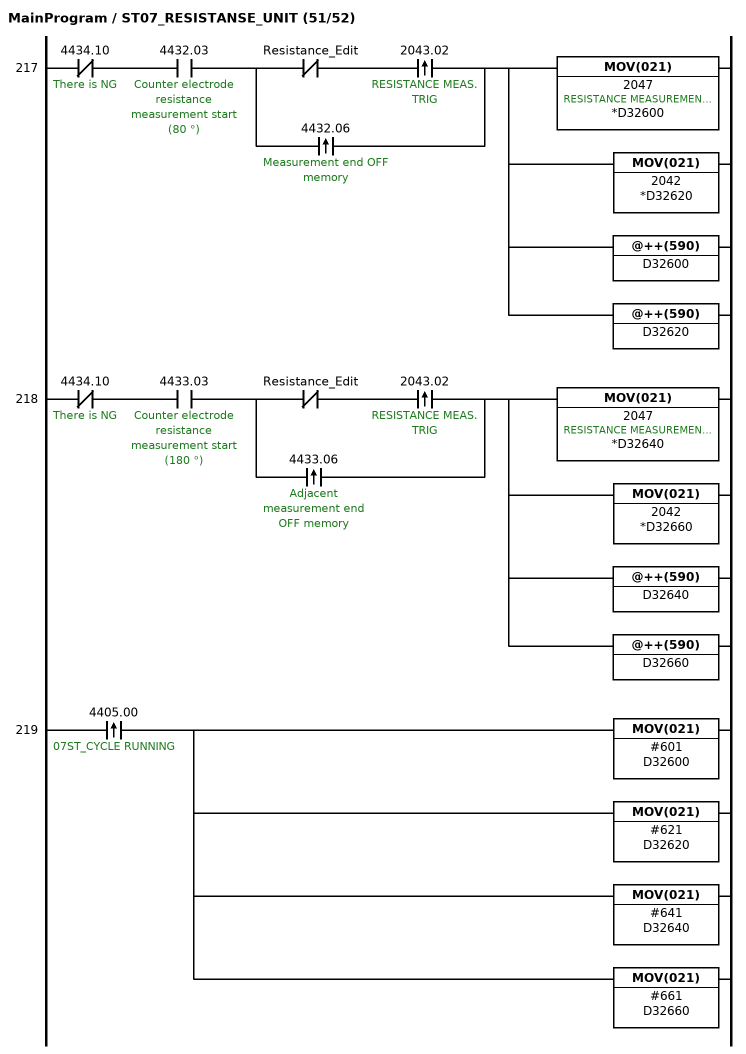
; rung 217
LDNOT 4434.10  ; There is NG
AND 4432.03  ; Counter electrode resistance measurement start (80 °)
LDNOT Resistance_Edit
@AND 2043.02  ; RESISTANCE MEAS. TRIG
@OR 4432.06  ; Measurement end OFF memory
ANDLD
MOV(021) 2047 *D32600  ; RESISTANCE MEASUREMENT CHANGE RELAY
MOV(021) 2042 *D32620
@++(590) D32600
@++(590) D32620
; rung 218
LDNOT 4434.10  ; There is NG
AND 4433.03  ; Counter electrode resistance measurement start (180 °)
LDNOT Resistance_Edit
@AND 2043.02  ; RESISTANCE MEAS. TRIG
@OR 4433.06  ; Adjacent measurement end OFF memory
ANDLD
MOV(021) 2047 *D32640  ; RESISTANCE MEASUREMENT CHANGE RELAY
MOV(021) 2042 *D32660
@++(590) D32640
@++(590) D32660
; rung 219
@LD 4405.00  ; 07ST_CYCLE RUNNING
MOV(021) #601 D32600
MOV(021) #621 D32620
MOV(021) #641 D32640
MOV(021) #661 D32660

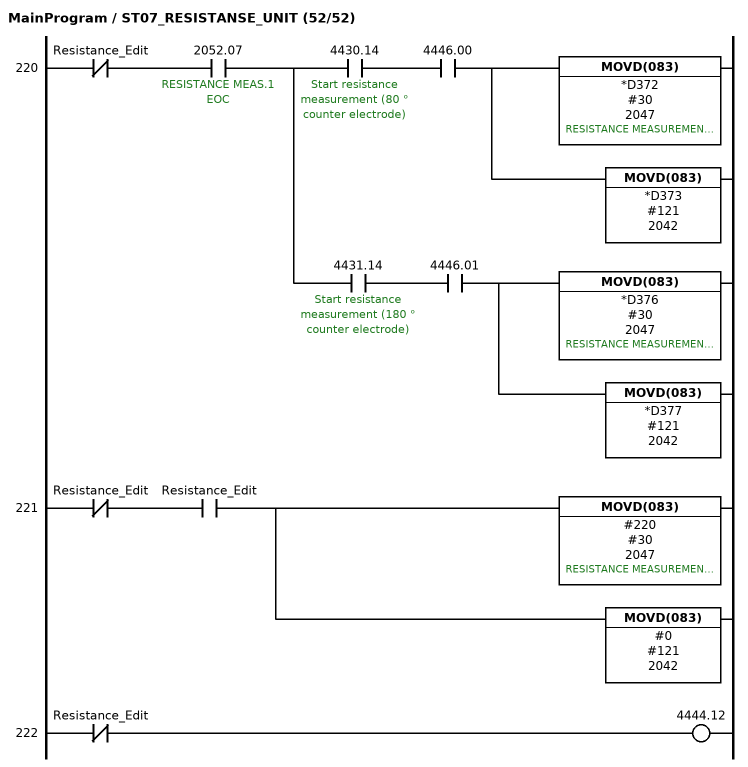
; rung 220
LDNOT Resistance_Edit
AND 2052.07  ; RESISTANCE MEAS.1 EOC
OUT TR0
AND 4430.14  ; Start resistance measurement (80 ° counter electrode)
AND 4446.00
MOVD(083) *D372 #30 2047  ; RESISTANCE MEASUREMENT CHANGE RELAY
MOVD(083) *D373 #121 2042
LD TR0
AND 4431.14  ; Start resistance measurement (180 ° counter electrode)
AND 4446.01
MOVD(083) *D376 #30 2047  ; RESISTANCE MEASUREMENT CHANGE RELAY
MOVD(083) *D377 #121 2042
; rung 221
LDNOT Resistance_Edit
AND Resistance_Edit
MOVD(083) #220 #30 2047  ; RESISTANCE MEASUREMENT CHANGE RELAY
MOVD(083) #0 #121 2042
; rung 222
LDNOT Resistance_Edit
OUT 4444.12
; rung 223: Data Feed

### Section ST08_IMPULSE_UNIT

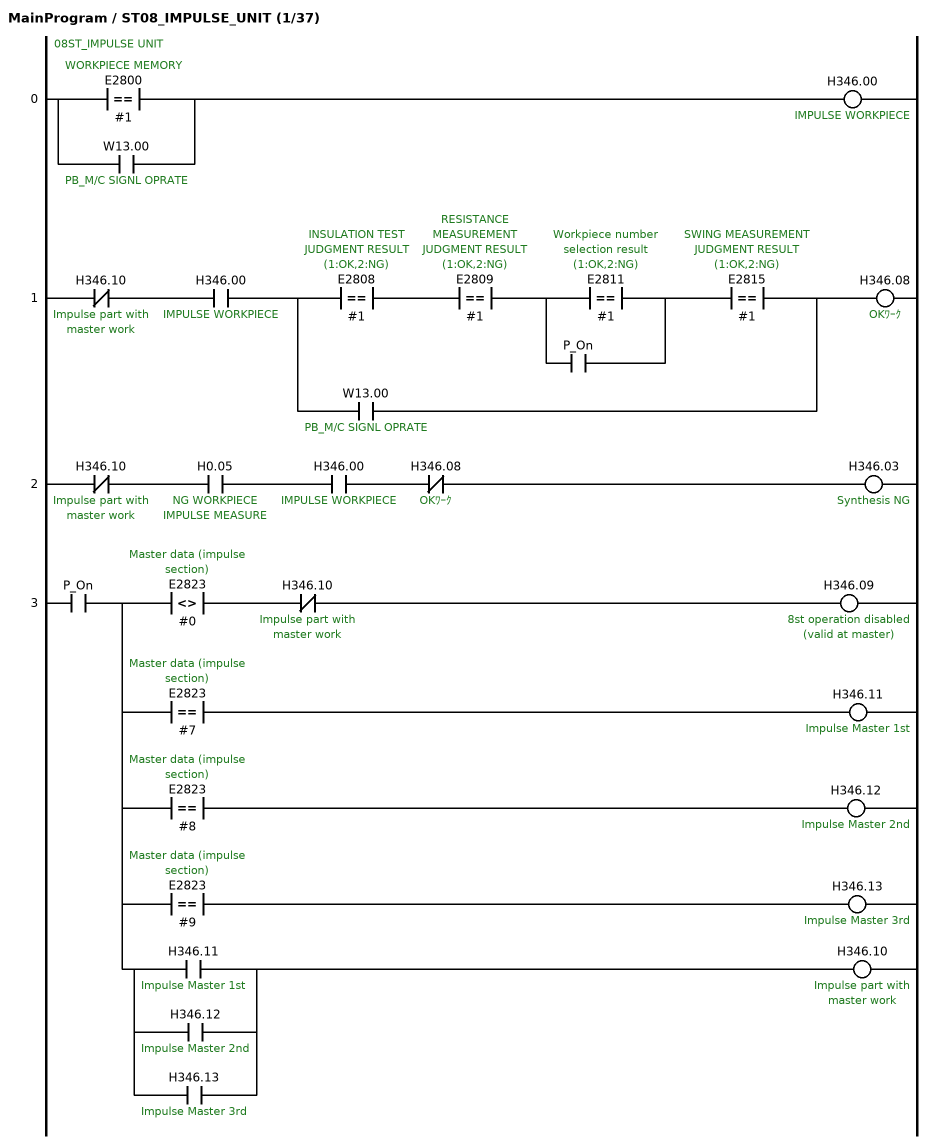
; rung 0: 08ST_IMPULSE UNIT
LD=(300) E2800 #1  ; WORKPIECE MEMORY
OR W13.00  ; PB_M/C SIGNL OPRATE
OUT H346.00  ; IMPULSE WORKPIECE
; rung 1
LDNOT H346.10  ; Impulse part with master work
AND H346.00  ; IMPULSE WORKPIECE
LD=(300) E2808 #1  ; INSULATION TEST JUDGMENT RESULT (1:OK,2:NG)
AND=(300) E2809 #1  ; RESISTANCE MEASUREMENT JUDGMENT RESULT (1:OK,2:NG)
LD=(300) E2811 #1  ; Workpiece number selection result (1:OK,2:NG)
OR P_On
ANDLD
AND=(300) E2815 #1  ; SWING MEASUREMENT JUDGMENT RESULT (1:OK,2:NG)
OR W13.00  ; PB_M/C SIGNL OPRATE
ANDLD
OUT H346.08  ; OKﾜｰｸ
; rung 2
LDNOT H346.10  ; Impulse part with master work
AND H0.05  ; NG WORKPIECE IMPULSE MEASURE
AND H346.00  ; IMPULSE WORKPIECE
ANDNOT H346.08  ; OKﾜｰｸ
OUT H346.03  ; Synthesis NG
; rung 3
LD P_On
OUT TR0
AND<>(305) E2823 #0  ; Master data (impulse section)
ANDNOT H346.10  ; Impulse part with master work
OUT H346.09  ; 8st operation disabled (valid at master)
LD TR0
AND=(300) E2823 #7  ; Master data (impulse section)
OUT H346.11  ; Impulse Master 1st
LD TR0
AND=(300) E2823 #8  ; Master data (impulse section)
OUT H346.12  ; Impulse Master 2nd
LD TR0
AND=(300) E2823 #9  ; Master data (impulse section)
OUT H346.13  ; Impulse Master 3rd
LD TR0
LD H346.11  ; Impulse Master 1st
OR H346.12  ; Impulse Master 2nd
OR H346.13  ; Impulse Master 3rd
ANDLD
OUT H346.10  ; Impulse part with master work

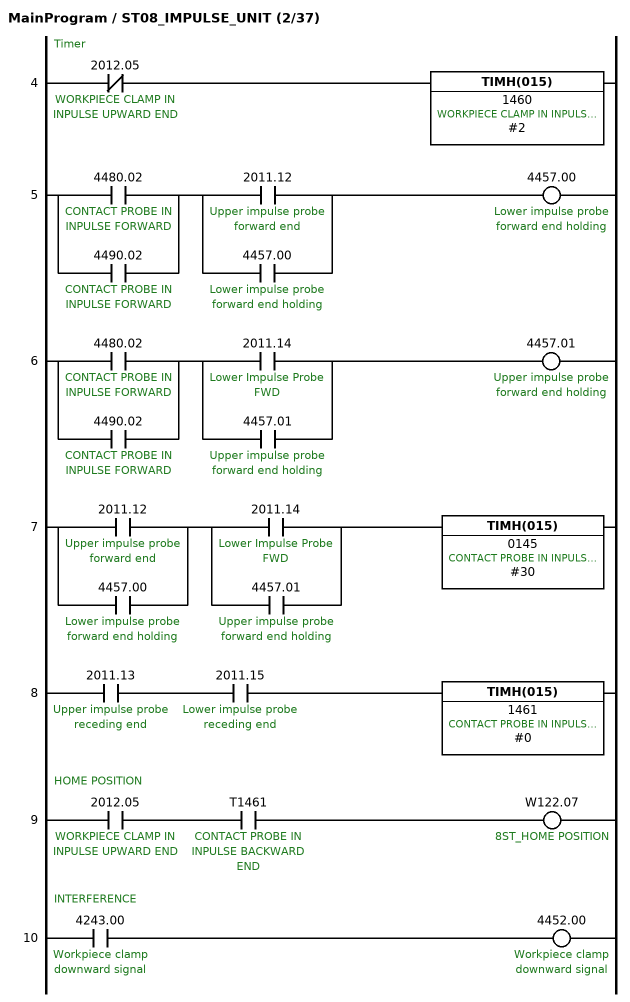
; rung 4: Timer
LDNOT 2012.05  ; WORKPIECE CLAMP IN INPULSE UPWARD END
TIMH(015) 1460 #2  ; WORKPIECE CLAMP IN INPULSE DOWNWARD END
; rung 5
LD 4480.02  ; CONTACT PROBE IN INPULSE FORWARD
OR 4490.02  ; CONTACT PROBE IN INPULSE FORWARD
LD 2011.12  ; Upper impulse probe forward end
OR 4457.00  ; Lower impulse probe forward end holding
ANDLD
OUT 4457.00  ; Lower impulse probe forward end holding
; rung 6
LD 4480.02  ; CONTACT PROBE IN INPULSE FORWARD
OR 4490.02  ; CONTACT PROBE IN INPULSE FORWARD
LD 2011.14  ; Lower Impulse Probe FWD
OR 4457.01  ; Upper impulse probe forward end holding
ANDLD
OUT 4457.01  ; Upper impulse probe forward end holding
; rung 7
LD 2011.12  ; Upper impulse probe forward end
OR 4457.00  ; Lower impulse probe forward end holding
LD 2011.14  ; Lower Impulse Probe FWD
OR 4457.01  ; Upper impulse probe forward end holding
ANDLD
TIMH(015) 0145 #30  ; CONTACT PROBE IN INPULSE FORWARD END
; rung 8
LD 2011.13  ; Upper impulse probe receding end
AND 2011.15  ; Lower impulse probe receding end
TIMH(015) 1461 #0  ; CONTACT PROBE IN INPULSE BACKWARD END  // #2 => #0
; rung 9: HOME POSITION
LD 2012.05  ; WORKPIECE CLAMP IN INPULSE UPWARD END
AND T1461  ; CONTACT PROBE IN INPULSE BACKWARD END
OUT W122.07  ; 8ST_HOME POSITION
; rung 10: INTERFERENCE
LD 4243.00  ; Workpiece clamp downward signal
OUT 4452.00  ; Workpiece clamp downward signal

